ABB RAPID module: SharedModule.mod

MODULE SharedModule(NOSTEPIN)
    !*****************************************************
    !Module Name:   SharedModule
    !Version:       1.0
    !Description:
    !Date:          2021-1-6
    !Author:        Michael
    !*****************************************************

    !2021-8-11, Michael, Add numScanJob1, ScanSeamByLaser, ScanData
    !2021-8-12, Michael, Add GetDropFeet
    !2021-8-13, Michael, Add ReloadGantryOffset
    !2021-8-16, Michael, Add RefreshDisplacement
    !2021-8-20, Michael, Add WriteSysDataLog

    RECORD ScanData
        num joint_no;
    ENDRECORD

    PERS string strTab:=",";
    PERS string strUtilityKey:="ZhongXun2021";

    !numJobMode: 0 - Keep last, 1 - by TPU, 2 - by yml, 3 - by PLC
    PERS num numJobMode:=2;

    !For numJobMode=1
    PERS RECORDModelData rModelDataFirst{4}:=[["30014",[-2155,0,60]],["",[-2155,0,60]],["",[-2155,0,60]],["",[-2155,0,60]]];
    PERS pos posModelOffset:=[-1670,10,0];
    PERS num numModelOffsetStart:=1;
    PERS num numModelOffsetQuantity:=1;

    !For numJobMode=3
    PERS dnum numPLCJobID:=1;
    PERS num numGantryPosition:=36;

    PROC MovetoHome()
        VAR jointtarget jointCur;
        EOffsOff;
        WHILE jointHome.robax<>jointHomeOld.robax DO
            UIMsgBox\Header:="Home Position Changed",""\MsgLine2:="Robot Home Position has been changed."\MsgLine3:="Please check it."\MsgLine4:="Restart the robot controller to update it."\Buttons:=btnOK\Icon:=iconWarning;
        ENDWHILE
        jointCur:=CJointT();
        jointHome.extax.eax_a:=jointCur.extax.eax_a;
        jointHome.extax.eax_b:=jointCur.extax.eax_b;
        !jointHome.extax.eax_c:=extGantryHome.eax_c;
        MoveAbsJ jointHome,speedAir,fine,toolWeldGun\WObj:=wobj0;
    ENDPROC

    PROC MoveToReadyQuadrant(num numQuadrant)
        VAR pos posGantryOffsetDirection:=[0,0,0];
        posGantryOffsetDirection:=GetGantryOffsetDirection(numQuadrant);
        TEST numQuadrant
        CASE 1:
            jointReadyQuadrant1.extax.eax_a:=extjointGantryOffset.eax_a*posGantryOffsetDirection.x;
            jointReadyQuadrant1.extax.eax_b:=extjointGantryOffset.eax_b*posGantryOffsetDirection.y;
            jointReadyQuadrant1.extax.eax_c:=jointHome.extax.eax_c-C_PROGDISP.eoffs.eax_c;
            jointCurrent:=jointReadyQuadrant1;
        CASE 2:
            jointReadyQuadrant2.extax.eax_a:=extjointGantryOffset.eax_a*posGantryOffsetDirection.x;
            jointReadyQuadrant2.extax.eax_b:=extjointGantryOffset.eax_b*posGantryOffsetDirection.y;
            jointReadyQuadrant2.extax.eax_c:=jointHome.extax.eax_c-C_PROGDISP.eoffs.eax_c;
            jointCurrent:=jointReadyQuadrant2;
        CASE 3:
            jointReadyQuadrant3.extax.eax_a:=extjointGantryOffset.eax_a*posGantryOffsetDirection.x;
            jointReadyQuadrant3.extax.eax_b:=extjointGantryOffset.eax_b*posGantryOffsetDirection.y;
            jointReadyQuadrant3.extax.eax_c:=jointHome.extax.eax_c-C_PROGDISP.eoffs.eax_c;
            jointCurrent:=jointReadyQuadrant3;
        CASE 4:
            jointReadyQuadrant4.extax.eax_a:=extjointGantryOffset.eax_a*posGantryOffsetDirection.x;
            jointReadyQuadrant4.extax.eax_b:=extjointGantryOffset.eax_b*posGantryOffsetDirection.y;
            jointReadyQuadrant4.extax.eax_c:=jointHome.extax.eax_c-C_PROGDISP.eoffs.eax_c;
            jointCurrent:=jointReadyQuadrant4;
        CASE 14:
            jointReadyQuadrant1.extax.eax_a:=extjointGantryOffset.eax_a*posGantryOffsetDirection.x;
            jointReadyQuadrant1.extax.eax_b:=extjointGantryOffset.eax_b*posGantryOffsetDirection.y;
            jointReadyQuadrant1.extax.eax_c:=jointHome.extax.eax_c-C_PROGDISP.eoffs.eax_c;
            jointCurrent:=jointReadyQuadrant1;
        CASE 23:
            jointReadyQuadrant2.extax.eax_a:=extjointGantryOffset.eax_a*posGantryOffsetDirection.x;
            jointReadyQuadrant2.extax.eax_b:=extjointGantryOffset.eax_b*posGantryOffsetDirection.y;
            jointReadyQuadrant2.extax.eax_c:=jointHome.extax.eax_c-C_PROGDISP.eoffs.eax_c;
            jointCurrent:=jointReadyQuadrant2;
        DEFAULT:
            RETURN ;
        ENDTEST
        MoveAbsJ jointCurrent,speedAir,zoneAir,toolWeldGun\WObj:=wobjCurrent;
    ENDPROC

    PROC Scan_1D_Laser(INOUT robtarget ScanFound,robtarget ScanPoint,num JointNo)
        Logging "Scan:"+ValToStr(ScanPoint.trans);
        MoveL ScanPoint,speedAproach,fine,toolLaser\WObj:=wobjCurrent;
        WaitTime numWaitTimeForLaser/2;
        IF RobOS() THEN
            ScanFound:=ScanPoint;
            Logging "Found:"+ValToStr(ScanFound.trans);
        ELSE
            ScanFound:=ScanPoint;
        ENDIF
    ENDPROC

    PROC ScanSeamByLaser(INOUT robtarget ScanFound,robtarget ScanPoint,ScanData JointData,speeddata Speed,PERS tooldata Tool\PERS wobjdata WObj)
        Logging "Scan: "+ArgName(ScanPoint)+"="+ValToStr(ScanPoint.trans);
        MoveJ ScanPoint,speedAproach,fine,Tool\WObj?WObj;
        WaitTime numWaitTimeForLaser/2;
        IF RobOS() THEN
            SeamFind JointData.joint_no\FoundPoint:=ScanFound,ScanPoint,speedAproach,js1,SenSch1,Tool\WObj?WObj;
        ELSE
            IF boolDebugSearch THEN
                UIMsgBox\Header:="Simulation Laser Sensor","Use scan point for found point"\MsgLine3:="Press OK to continue"\Buttons:=btnOK\Icon:=iconWarning;
            ENDIF
            ScanFound:=ScanPoint;
        ENDIF
        Logging "Found: "+ArgName(ScanFound)+"="+ValToStr(ScanFound.trans);
    ENDPROC

    PROC UpdateWeldSeamStatus(\switch Start,num numSeamIndex)
        VAR dnum dnumWeldSeamStatus;
        dnumWeldSeamStatus:=GOutputDnum(Go112_WeldCompleted);
        IF Present(Start) THEN
            BitClear dnumWeldSeamStatus,numSeamIndex;
            SetGO Go112_WeldCompleted,dnumWeldSeamStatus;

            SetGO Go80_WeldingStatus,PowDnum(2,numSeamIndex-1);
        ELSE
            SetGO Go80_WeldingStatus,0;

            BitSet dnumWeldSeamStatus,numSeamIndex;
            SetGO Go112_WeldCompleted,dnumWeldSeamStatus;
        ENDIF
    ENDPROC

    PROC LoadModelDatabyTPU()
        VAR num numIndex:=0;
        Logging "Offset: "+ValToStr(posModelOffset);
        Logging "Quantity: "+ValToStr(numModelOffsetQuantity);
        FOR i FROM numModelOffsetStart TO numModelOffsetQuantity DO
            FOR j FROM 1 TO Dim(rModelDataFirst,1) DO
                IF rModelDataFirst{j}.name<>"" THEN
                    Incr numIndex;
                    Logging "Load: "+ValToStr(rModelDataFirst{j}.name);
                    strWeldPartList{numIndex}:=rModelDataFirst{j}.name;
                    posWeldPartList{numIndex}:=rModelDataFirst{j}.location+posModelOffset*(i-1);
                ENDIF
            ENDFOR
        ENDFOR
        numModelStart:=1;
        numModelQuantity:=numModelOffsetQuantity-numModelOffsetStart+1;
    ENDPROC

    PROC LoadModelDatabyYML()
        VAR num numIndex:=0;
        Logging "LoadModelDatabyYML";
        LoadModelDataYamlFile strModelDataYamlFileName;
        FOR i FROM 1 TO Dim(rModelDataArray,1) DO
            IF rModelDataArray{i}.name<>"" THEN
                Incr numIndex;
                Logging "Load: "+ValToStr(rModelDataArray{i}.name);
                strWeldPartList{numIndex}:=rModelDataArray{i}.name;
                posWeldPartList{numIndex}:=rModelDataArray{i}.location;
            ENDIF
        ENDFOR
        numModelStart:=1;
        numModelQuantity:=numIndex;
    ENDPROC

    PROC LoadModelDatabyPLC()
        Logging "LoadModelDatabyPLC";
        numPLCJobID:=GInputDnum(Gi112_JobID);
        numGantryPosition:=AInput(Ai144_GantryPosition);
        Logging "numPLCJobID="+ValToStr(numPLCJobID);
        Logging "numGantryPosition="+ValToStr(numGantryPosition);
        strModelDataYamlFileName:="job_"+ValToStr(numPLCJobID)+".yml";
        LoadModelDatabyYML;
    ENDPROC

    PROC InhibWeld(bool boolInhib\switch Weld\switch Weave\switch Track)
        IF boolInhib THEN
            IF Present(Weave) THEN
                SetDO sdoWeldInhib,1;
            ENDIF
            IF Present(Weave) THEN
                SetDO sdoWeldInhib,1;
            ENDIF
            IF Present(Track) THEN
                SetDO sdoTrackInhib,1;
            ENDIF
        ELSE
            IF Present(Weave) THEN
                SetDO sdoWeldInhib,0;
            ENDIF
            IF Present(Weave) THEN
                SetDO sdoWeldInhib,0;
            ENDIF
            IF Present(Track) THEN
                SetDO sdoTrackInhib,0;
            ENDIF
        ENDIF
    ENDPROC

    PROC WriteSysDataLog(string strTemplateID)
        Close iodevSysDataLog;
        IF boolInitSysDataLogFile THEN
            Open "HOME:"\File:=strSysDataLogFileName,iodevSysDataLog;
            Write iodevSysDataLog,"Time"+strTab+"TemplateID"\NoNewLine;
            Write iodevSysDataLog,strTab+"WeldGun.X"+strTab+"WeldGun.Y"+strTab+"WeldGun.Z"\NoNewLine;
            Write iodevSysDataLog,strTab+"WeldGun.Orient"\NoNewLine;
            Write iodevSysDataLog,strTab+"uframe.X"+strTab+"uframe.Y"+strTab+"uframe.Z"\NoNewLine;
            Write iodevSysDataLog,strTab+"uframe.Orient"\NoNewLine;
            Write iodevSysDataLog,strTab+"oframe.X"+strTab+"oframe.Y"+strTab+"oframe.Z"\NoNewLine;
            Write iodevSysDataLog,strTab+"oframe.Orient";
            boolInitSysDataLogFile:=FALSE;
        ELSE
            Open "HOME:"\File:=strSysDataLogFileName,iodevSysDataLog\Append;
        ENDIF
        Write iodevSysDataLog,CDate()+" "+CTime()+strTab+strTemplateID\NoNewLine;
        Write iodevSysDataLog,strTab+ValToStr(toolWeldGun.tframe.trans.x)+strTab+ValToStr(toolWeldGun.tframe.trans.y)+strTab+ValToStr(toolWeldGun.tframe.trans.z)\NoNewLine;
        Write iodevSysDataLog,strTab+EncapsulateString(GetEulerAngleString(toolWeldGun.tframe.rot))\NoNewLine;
        Write iodevSysDataLog,strTab+ValToStr(wobjCurrent.uframe.trans.x)+strTab+ValToStr(wobjCurrent.uframe.trans.y)+strTab+ValToStr(wobjCurrent.uframe.trans.z)\NoNewLine;
        Write iodevSysDataLog,strTab+EncapsulateString(GetEulerAngleString(wobjCurrent.uframe.rot))\NoNewLine;
        Write iodevSysDataLog,strTab+ValToStr(wobjCurrent.oframe.trans.x)+strTab+ValToStr(wobjCurrent.oframe.trans.y)+strTab+ValToStr(wobjCurrent.oframe.trans.z)\NoNewLine;
        Write iodevSysDataLog,strTab+EncapsulateString(GetEulerAngleString(wobjCurrent.oframe.rot));
        Close iodevSysDataLog;
        Logging "WriteSysDataLog is done";
    ENDPROC

ENDMODULE
